{attribute addProperty BoxType "EL2521-0000-1016"}
{attribute addProperty Id "PTO_StatusAT %I*PTO_Status_CB1E42AE5670ENC_Status_compactAT %I*ENC_Status_compact_D18EAE2D5670PTO_ControlAT %Q*PTO_Control_DFE022934050PTO_Target_compactAT %Q*PTO_Target_compact_C80C22BB1620ENC_Control_compactAT %Q*ENC_Control_compact_8FDE73942430WcStateAT %I*WcState_98A4DF7520.250InfoDataAT %I*InfoData_BC63D37F80100"}
{attribute addProperty CRC "435489933"}
{attribute addProperty SizeInBites "274"}
{attribute addProperty SizeInBytes "34.25"}
TYPE EL2521_54A6CFE2 :
STRUCT
	{attribute addProperty Name "PTO_Status"}
	PTO_Status : PTO_Status_CB1E42AE;
	{attribute addProperty Name "ENC_Status_compact"}
	ENC_Status_compact : ENC_Status_compact_D18EAE2D;
	{attribute addProperty Name "PTO_Control"}
	PTO_Control : PTO_Control_DFE02293;
	{attribute addProperty Name "PTO_Target_compact"}
	PTO_Target_compact : PTO_Target_compact_C80C22BB;
	{attribute addProperty Name "ENC_Control_compact"}
	ENC_Control_compact : ENC_Control_compact_8FDE7394;
	{attribute addProperty Name "WcState"}
	WcState : WcState_98A4DF75;
	{attribute addProperty Name "InfoData"}
	InfoData : InfoData_BC63D37F;
END_STRUCT
END_TYPE

(* stored: Version 1.2.0.0, ProductVersion 3.1.4024.9
   DUT EL2521_54A6CFE2: Id {19085158-7c78-4372-ba27-c482eb5cb978} *)
